PROGRAM UPTIME
VAR
	timeInit : BOOL :=TRUE;
	Timer : TON;
	time1 : TIME;
	time2 : TIME;
	{attribute 'OPC.UA.DA' :='1'}
	Eng : EngStruct;
	
END_VAR

Timer(IN := timeInit, PT := T#5S);

IF timeInit THEN
	time1 := TIME();
	timeInit := FALSE;
END_IF

	time2 := TIME();

Eng.uptime := time_to_string(time2-time1);

END_PROGRAM

(* stored: Version 1.1.0.1, ProductVersion 3.1.4024.10
   POU UPTIME: Id {7357bad6-cff8-41e1-9f32-3618f1446314}, SpecialFunc None *)
